{attribute 'qualified_only'}
VAR_GLOBAL
END_VAR

(* stored: Version 1.1.0.1, ProductVersion 3.1.4024.12
   GVL GVL: Id {84bc136a-4fc0-4d0a-9eb7-e638f4d7660b} *)
